FUNCTION_BLOCK "FB_SimpleBlockWithInputs"

   VAR_INPUT
        IN : DINT;
   END_VAR

   VAR_OUTPUT
        OUT : DINT;
   END_VAR

   VAR
        otherVar1 : DINT;
   END_VAR

BEGIN

END_FUNCTION_BLOCK